PROGRAM P_Demo_DT_TO_SYSTEMTIME
VAR
    dtCurrent : DATE_AND_TIME := DT#2026-05-11-12:34:56; // 当前 PLC 时间（来自 F_GetActualDateTime）
    stCurrent : TIMESTRUCT; // 转换后的系统时间结构（HMI 绑定字段）
    bRunOnce  : BOOL; // 脉冲触发一次执行
END_VAR

// =============================================================================
// 场景：HMI 显示当前 PLC 时间需按 年-月-日-时-分-秒 拆分字段
//
// 价值：1 行调用拿到 7 个时间字段（自动算 wDayOfWeek），不用手写整除取余
//
// 验证步骤：
//   1. 引用 Tc2_Utilities
//   2. 编译 + 登录 + 运行
//   3. 强制 bRunOnce := TRUE 一个周期
//   4. 在线监视 stCurrent.wYear=2026, wMonth=5, wDay=11, wHour=12, wMinute=34, wSecond=56
//   5. 注意 wMilliseconds 永远为 0（DT 精度只到秒）
// =============================================================================
stCurrent := DT_TO_SYSTEMTIME(dtCurrent);

END_PROGRAM

(* stored: Version 1.1.0.1, ProductVersion 3.1.4024.5
   POU P_Demo_DT_TO_SYSTEMTIME: Id {bd539bb1-96e6-52b2-8d92-28dabda3c0a5}, SpecialFunc None *)
